// TIA Portal V19 export
DATA_BLOCK "Analogwerte"   // DB1110
{ S7_Optimized_Access := 'TRUE' }
// stored: AutoNumber false, MemoryReserve 100
   VAR RETAIN
      "LF_CM01.BN01" : Struct   // Leitfähigkeit Bypass Filterpumpe
         MB_min : Real := 0.0;
         MB_max : Real := 2000.0;   // mS
         UG_Alarm : Real := -0.5;
         OG_Alarm : Real := 2200.0;
         GF : Real := 0.5;
         Drahtbruch : Bool := FALSE;
         ungueltig : Bool := FALSE;
      END_STRUCT;
      "LF_CM01.BN02" : Struct   // Leitfähigkeit Düsen Umwälzung
         MB_min : Real := 0.0;
         MB_max : Real := 2000.0;   // mS
         UG_Alarm : Real := -0.5;
         OG_Alarm : Real := 2200.0;
         GF : Real := 0.5;
         Drahtbruch : Bool := FALSE;
         ungueltig : Bool := FALSE;
      END_STRUCT;
      "LF_CM02.BN03" : Struct   // Leitfähigkeit Bypass Filterpumpe
         MB_min : Real := 0.0;
         MB_max : Real := 2000.0;   // mS
         UG_Alarm : Real := -0.5;
         OG_Alarm : Real := 2200.0;
         GF : Real := 0.5;
         Drahtbruch : Bool := FALSE;
         ungueltig : Bool := FALSE;
      END_STRUCT;
      "LF_CM02.BN04" : Struct   // Leitfähigkeit Düsen Umwälzung
         MB_min : Real := 0.0;
         MB_max : Real := 2000.0;   // mS
         UG_Alarm : Real := -0.5;
         OG_Alarm : Real := 2200.0;
         GF : Real := 0.5;
         Drahtbruch : Bool := FALSE;
         ungueltig : Bool := FALSE;
      END_STRUCT;
      "p_HQ01.BP01" : Struct   // Druck Beutelfiltergehäuse
         MB_min : Real := 0.0;
         MB_max : Real := 4.0;   // bar
         UG_Alarm : Real := -0.5;
         OG_Alarm : Real := 4.5;
         GF : Real := 0.5;
         Drahtbruch : Bool := FALSE;
         ungueltig : Bool := FALSE;
      END_STRUCT;
      "p_HQ02.BP02" : Struct   // Druck Beutelfiltergehäuse
         MB_min : Real := 0.0;
         MB_max : Real := 4.0;   // bar
         UG_Alarm : Real := -0.5;
         OG_Alarm : Real := 4.5;
         GF : Real := 0.5;
         Drahtbruch : Bool := FALSE;
         ungueltig : Bool := FALSE;
      END_STRUCT;
      "p_CM01.BP03" : Struct   // Druck Filterpumpe
         MB_min : Real := 0.0;
         MB_max : Real := 4.0;   // bar
         UG_Alarm : Real := -0.5;
         OG_Alarm : Real := 4.5;
         GF : Real := 0.5;
         Drahtbruch : Bool := FALSE;
         ungueltig : Bool := FALSE;
      END_STRUCT;
      "p_CM01.BP04" : Struct   // Druck Umwälzpumpe
         MB_min : Real := 0.0;
         MB_max : Real := 4.0;   // bar
         UG_Alarm : Real := -0.5;
         OG_Alarm : Real := 4.5;
         GF : Real := 0.5;
         Drahtbruch : Bool := FALSE;
         ungueltig : Bool := FALSE;
      END_STRUCT;
      "p_CM03.BP05" : Struct   // Druck Umwäzpumpe
         MB_min : Real := 0.0;
         MB_max : Real := 4.0;   // bar
         UG_Alarm : Real := -0.5;
         OG_Alarm : Real := 4.5;
         GF : Real := 0.5;
         Drahtbruch : Bool := FALSE;
         ungueltig : Bool := FALSE;
      END_STRUCT;
      "p_CM02.BP06" : Struct   // Druck Filterpumpe
         MB_min : Real := 0.0;
         MB_max : Real := 4.0;   // bar
         UG_Alarm : Real := -0.5;
         OG_Alarm : Real := 4.5;
         GF : Real := 0.5;
         Drahtbruch : Bool := FALSE;
         ungueltig : Bool := FALSE;
      END_STRUCT;
      "p_CM02.BP07" : Struct   // Druck Umwälzpumpe
         MB_min : Real := 0.0;
         MB_max : Real := 4.0;   // bar
         UG_Alarm : Real := -0.5;
         OG_Alarm : Real := 4.5;
         GF : Real := 0.5;
         Drahtbruch : Bool := FALSE;
         ungueltig : Bool := FALSE;
      END_STRUCT;
      "p_CM04.BP08" : Struct   // Druck Umwäzpumpe
         MB_min : Real := 0.0;
         MB_max : Real := 4.0;   // bar
         UG_Alarm : Real := -0.5;
         OG_Alarm : Real := 4.5;
         GF : Real := 0.5;
         Drahtbruch : Bool := FALSE;
         ungueltig : Bool := FALSE;
      END_STRUCT;
      "p_CM05.BP09" : Struct   // Druck Pumpe Entleerung Sammeltank
         MB_min : Real := 0.0;
         MB_max : Real := 4.0;   // bar
         UG_Alarm : Real := -0.5;
         OG_Alarm : Real := 4.5;
         GF : Real := 0.5;
         Drahtbruch : Bool := FALSE;
         ungueltig : Bool := FALSE;
      END_STRUCT;
      "Dfl_GP01.BF01" : Struct   // Durchfluss Versorgung Frischsäure
         MB_min : Real := 0.0;
         MB_max : Real := 2000.0;   // ml/s
         UG_Alarm : Real := -0.5;
         OG_Alarm : Real := 2200.0;
         GF : Real := 0.5;
         Drahtbruch : Bool := FALSE;
         ungueltig : Bool := FALSE;
      END_STRUCT;
      "Dfl_GP02.BF02" : Struct   // Durchfluss Entsorgung Altsäure
         MB_min : Real := 0.0;
         MB_max : Real := 2000.0;   // ml/s
         UG_Alarm : Real := -0.5;
         OG_Alarm : Real := 2200.0;
         GF : Real := 0.5;
         Drahtbruch : Bool := FALSE;
         ungueltig : Bool := FALSE;
      END_STRUCT;
      "Niv_GP01.BL30" : Struct   // Füllstand Versorgung Frischsäure
         MB_min : Real := 0.0;
         MB_max : Real := 100.0;   // %
         UG_Alarm : Real := -0.5;
         OG_Alarm : Real := 110.0;
         GF : Real := 0.5;
         Drahtbruch : Bool := FALSE;
         ungueltig : Bool := FALSE;
      END_STRUCT;
      "Niv_GP02.BL31" : Struct   // Füllstand Entsorgung Altsäure
         MB_min : Real := 0.0;
         MB_max : Real := 100.0;   // %
         UG_Alarm : Real := -0.5;
         OG_Alarm : Real := 110.0;
         GF : Real := 0.5;
         Drahtbruch : Bool := FALSE;
         ungueltig : Bool := FALSE;
      END_STRUCT;
      pH_WR01 : Struct   // pH-Wert Be-/Entladen
         MB_min : Real := 0.0;
         MB_max : Real := 100.0;   // %
         UG_Alarm : Real := -0.5;
         OG_Alarm : Real := 110.0;
         GF : Real := 0.5;
         Drahtbruch : Bool := FALSE;
         ungueltig : Bool := FALSE;
      END_STRUCT;
      WZ_1_1 : Struct   // Wägezelle WR04.BW01
         MB_min : Real := 0.0;
         MB_max : Real := 100.0;   // %
         UG_Alarm : Real := -0.5;
         OG_Alarm : Real := 110.0;
         GF : Real := 0.5;
         Drahtbruch : Bool := FALSE;
         ungueltig : Bool := FALSE;
      END_STRUCT;
      WZ_1_2 : Struct   // Wägezelle WR04.BW02
         MB_min : Real := 0.0;
         MB_max : Real := 100.0;   // %
         UG_Alarm : Real := -0.5;
         OG_Alarm : Real := 110.0;
         GF : Real := 0.5;
         Drahtbruch : Bool := FALSE;
         ungueltig : Bool := FALSE;
      END_STRUCT;
      WZ_1_3 : Struct   // Wägezelle WR04.BW03
         MB_min : Real := 0.0;
         MB_max : Real := 100.0;   // %
         UG_Alarm : Real := -0.5;
         OG_Alarm : Real := 110.0;
         GF : Real := 0.5;
         Drahtbruch : Bool := FALSE;
         ungueltig : Bool := FALSE;
      END_STRUCT;
      WZ_1_4 : Struct   // Wägezelle WR04.BW04
         MB_min : Real := 0.0;
         MB_max : Real := 100.0;   // %
         UG_Alarm : Real := -0.5;
         OG_Alarm : Real := 110.0;
         GF : Real := 0.5;
         Drahtbruch : Bool := FALSE;
         ungueltig : Bool := FALSE;
      END_STRUCT;
      WZ_2_1 : Struct   // Wägezelle WR05.BW01
         MB_min : Real := 0.0;
         MB_max : Real := 100.0;   // %
         UG_Alarm : Real := -0.5;
         OG_Alarm : Real := 110.0;
         GF : Real := 0.5;
         Drahtbruch : Bool := FALSE;
         ungueltig : Bool := FALSE;
      END_STRUCT;
      WZ_2_2 : Struct   // Wägezelle WR05.BW01
         MB_min : Real := 0.0;
         MB_max : Real := 100.0;   // %
         UG_Alarm : Real := -0.5;
         OG_Alarm : Real := 110.0;
         GF : Real := 0.5;
         Drahtbruch : Bool := FALSE;
         ungueltig : Bool := FALSE;
      END_STRUCT;
      WZ_2_3 : Struct   // Wägezelle WR05.BW01
         MB_min : Real := 0.0;
         MB_max : Real := 100.0;   // %
         UG_Alarm : Real := -0.5;
         OG_Alarm : Real := 110.0;
         GF : Real := 0.5;
         Drahtbruch : Bool := FALSE;
         ungueltig : Bool := FALSE;
      END_STRUCT;
      WZ_2_4 : Struct   // Wägezelle WR05.BW01
         MB_min : Real := 0.0;
         MB_max : Real := 100.0;   // %
         UG_Alarm : Real := -0.5;
         OG_Alarm : Real := 110.0;
         GF : Real := 0.5;
         Drahtbruch : Bool := FALSE;
         ungueltig : Bool := FALSE;
      END_STRUCT;
      Last_1 : Struct   // Novamat WR04.BW34
         MB_min : Real := 0.0;
         MB_max : Real := 100.0;   // %
         UG_Alarm : Real := -0.5;
         OG_Alarm : Real := 110.0;
         GF : Real := 0.5;
         Drahtbruch : Bool := FALSE;
         ungueltig : Bool := FALSE;
      END_STRUCT;
      Last_2 : Struct   // Novamat WR05.BW43
         MB_min : Real := 0.0;
         MB_max : Real := 100.0;   // %
         UG_Alarm : Real := -0.5;
         OG_Alarm : Real := 110.0;
         GF : Real := 0.5;
         Drahtbruch : Bool := FALSE;
         ungueltig : Bool := FALSE;
      END_STRUCT;
   END_VAR
BEGIN
END_DATA_BLOCK
